FUNCTION_BLOCK FB_TEST3
VAR_INPUT
	execute: BOOL;
	pos2: LREAL := 2500;
END_VAR
VAR
	TIMERDONE: BOOL;
END_VAR

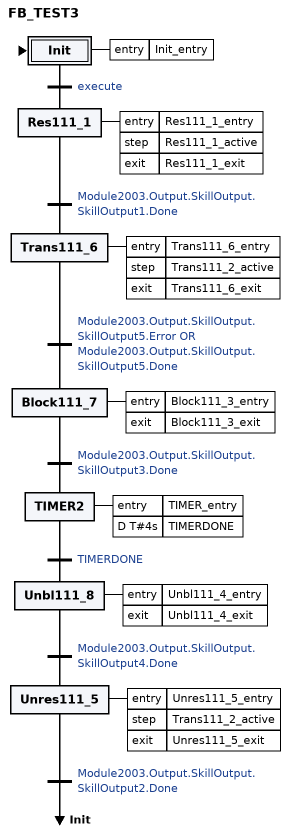
INITIAL_STEP Init:
    Init_entry(P1);  // entry action
END_STEP
TRANSITION FROM Init TO Res111_1
    := execute;
END_TRANSITION
STEP Res111_1:
    Res111_1_entry(P1);  // entry action
    Res111_1_active(N);  // step action
    Res111_1_exit(P0);  // exit action
END_STEP
TRANSITION FROM Res111_1 TO Trans111_6
    := Module2003.Output.SkillOutput.SkillOutput1.Done;
END_TRANSITION
STEP Trans111_6:
    Trans111_6_entry(P1);  // entry action
    Trans111_2_active(N);  // step action
    Trans111_6_exit(P0);  // exit action
END_STEP
TRANSITION FROM Trans111_6 TO Block111_7
    := Module2003.Output.SkillOutput.SkillOutput5.Error OR Module2003.Output.SkillOutput.SkillOutput5.Done;
END_TRANSITION
STEP Block111_7:
    Block111_3_entry(P1);  // entry action
    Block111_3_exit(P0);  // exit action
END_STEP
TRANSITION FROM Block111_7 TO TIMER2
    := Module2003.Output.SkillOutput.SkillOutput3.Done;
END_TRANSITION
STEP TIMER2:
    TIMER_entry(P1);  // entry action
    TIMERDONE(D, T#4s);
END_STEP
TRANSITION FROM TIMER2 TO Unbl111_8
    := TIMERDONE;
END_TRANSITION
STEP Unbl111_8:
    Unbl111_4_entry(P1);  // entry action
    Unbl111_4_exit(P0);  // exit action
END_STEP
TRANSITION FROM Unbl111_8 TO Unres111_5
    := Module2003.Output.SkillOutput.SkillOutput4.Done;
END_TRANSITION
STEP Unres111_5:
    Unres111_5_entry(P1);  // entry action
    Trans111_2_active(N);  // step action
    Unres111_5_exit(P0);  // exit action
END_STEP
TRANSITION FROM Unres111_5 TO Init
    := Module2003.Output.SkillOutput.SkillOutput2.Done;
END_TRANSITION

ACTION Trans111_6_exit:
//TRANSPORTIEREN

Module2003.Input.SkillInput.SkillInput5.Execute := FALSE;
Module2003.Input.SkillInput.SkillInput5.ParameterInput.Parameterinput1.Value := 0; //X-Position
Module2003.Input.SkillInput.SkillInput5.ParameterInput.Parameterinput2.Value := 0; //Z-Position
Module2003.Input.SkillInput.SkillInput5.ParameterInput.Parameterinput3.Value := 0; //Velocity
Module2003.Input.SkillInput.SkillInput5.ParameterInput.Parameterinput4.Value := 0; //Acceleration
END_ACTION

ACTION Res111_1_entry:
// Reservieren entry
Module2003.Input.SkillInput.SkillInput1.Execute := TRUE;
Module2003.Input.SkillInput.SkillInput1.ParameterInput.Parameterinput1.Value := 113; //TASKID
END_ACTION

ACTION Res111_1_active:

END_ACTION

ACTION Res111_1_exit:
// Reservieren entry
Module2003.Input.SkillInput.SkillInput1.Execute := FALSE;
Module2003.Input.SkillInput.SkillInput1.ParameterInput.Parameterinput1.Value := 0; //TASKID
END_ACTION

ACTION TIMER_entry:
TIMERDONE := FALSE;
END_ACTION

ACTION Trans111_6_entry:
//TRANSPORTIEREN

Module2003.Input.SkillInput.SkillInput5.Execute := TRUE;
Module2003.Input.SkillInput.SkillInput5.ParameterInput.Parameterinput1.Value := 2800; //X-Position
Module2003.Input.SkillInput.SkillInput5.ParameterInput.Parameterinput2.Value := 80; //Z-Position
Module2003.Input.SkillInput.SkillInput5.ParameterInput.Parameterinput3.Value := 0; //Velocity
Module2003.Input.SkillInput.SkillInput5.ParameterInput.Parameterinput4.Value := 0; //Acceleration
END_ACTION

ACTION Unbl111_4_exit:
//unBLOCKIEREN

Module2003.Input.SkillInput.SkillInput4.Execute := FALSE; 
Module2003.Input.SkillInput.SkillInput4.ParameterInput.Parameterinput1.Value := 000; //TaskID
END_ACTION

ACTION Trans111_2_entry:
//TRANSPORTIEREN

Module2003.Input.SkillInput.SkillInput5.Execute := TRUE;
Module2003.Input.SkillInput.SkillInput5.ParameterInput.Parameterinput1.Value := 2400; //X-Position
Module2003.Input.SkillInput.SkillInput5.ParameterInput.Parameterinput2.Value := 0; //Z-Position
Module2003.Input.SkillInput.SkillInput5.ParameterInput.Parameterinput3.Value := 300; //Velocity
Module2003.Input.SkillInput.SkillInput5.ParameterInput.Parameterinput4.Value := 100; //Acceleration
END_ACTION

ACTION Trans111_2_active:

END_ACTION

ACTION Unres111_5_exit:
//unreserve
Module2003.Input.SkillInput.SkillInput2.Execute := FALSE;
Module2003.Input.SkillInput.SkillInput2.ParameterInput.Parameterinput1.Value := 0; //TaskID
END_ACTION

ACTION Init_entry:
execute := FALSE;
END_ACTION

ACTION Trans111_2_exit:
//TRANSPORTIEREN

Module2003.Input.SkillInput.SkillInput5.Execute := FALSE;
Module2003.Input.SkillInput.SkillInput5.ParameterInput.Parameterinput1.Value := 0; //X-Position
Module2003.Input.SkillInput.SkillInput5.ParameterInput.Parameterinput2.Value := 0; //Z-Position
Module2003.Input.SkillInput.SkillInput5.ParameterInput.Parameterinput3.Value := 0; //Velocity
Module2003.Input.SkillInput.SkillInput5.ParameterInput.Parameterinput4.Value := 0; //Acceleration
END_ACTION

ACTION Block111_3_entry:
//BLOCKIEREN

Module2003.Input.SkillInput.SkillInput3.Execute := TRUE;
Module2003.Input.SkillInput.SkillInput3.ParameterInput.Parameterinput1.Value := 113; //TaskID
END_ACTION

ACTION Unres111_5_entry:
//unreserve
Module2003.Input.SkillInput.SkillInput2.Execute := TRUE;
Module2003.Input.SkillInput.SkillInput2.ParameterInput.Parameterinput1.Value := 113; //TaskID
END_ACTION

ACTION Block111_3_exit:
//BLOCKIEREN

Module2003.Input.SkillInput.SkillInput3.Execute := FALSE;
Module2003.Input.SkillInput.SkillInput3.ParameterInput.Parameterinput1.Value := 0; //TaskID
END_ACTION

ACTION Unbl111_4_entry:
//unBLOCKIEREN

Module2003.Input.SkillInput.SkillInput4.Execute := TRUE; //FALSE weil timer
Module2003.Input.SkillInput.SkillInput4.ParameterInput.Parameterinput1.Value := 112; //TaskID
END_ACTION

END_FUNCTION_BLOCK

(* stored: Version 1.1.0.1, ProductVersion 3.1.0.25
   POU FB_TEST3: Id {82879eaa-ab76-40c0-949a-0cc13c3506a3}
   Action Trans111_6_exit: Id {1b55c7e7-aa4e-405e-aa25-57a7c106dd22}
   Action Res111_1_entry: Id {320f2803-ca7d-4efc-aa52-c1728f991e0e}
   Action Res111_1_active: Id {4d2666ba-2187-42f1-b75d-b801821f9a8a}
   Action Res111_1_exit: Id {545a7478-02d9-44f3-8426-f9804fffc0a0}
   Action TIMER_entry: Id {7b0af5c3-2012-42fc-b13d-dba35455c33f}
   Action Trans111_6_entry: Id {80c10e71-f522-4b7c-8359-3a6de3697eda}
   Action Unbl111_4_exit: Id {858117a5-e6ff-4251-afd5-8491f453281e}
   Action Trans111_2_entry: Id {9146a7a3-75be-4ed5-aad1-f2b724c9c9db}
   Action Trans111_2_active: Id {99ba4a4c-ea55-42fc-acea-cdad15e7ab02}
   Action Unres111_5_exit: Id {9d6efc8c-8389-4c51-8571-6e0baf7122d3}
   Action Init_entry: Id {a19a2367-065b-475a-8daa-e73dd1c277c5}
   Action Trans111_2_exit: Id {ae315ed9-e17e-420a-b0f0-cbd2094bc820}
   Action Block111_3_entry: Id {b24f3b53-2f42-44cf-98fb-c35a24681cfd}
   Action Unres111_5_entry: Id {bb138fe8-fb53-4f09-8358-7c2ec9c29bb3}
   Action Block111_3_exit: Id {f20c18aa-4ad8-4308-97e2-e11249acc257}
   Action Unbl111_4_entry: Id {fe2f92e1-9508-4e7d-b6e8-8e402937af9f} *)
